// TIA Portal V20 export
DATA_BLOCK "IdentMvInterfaceHmi"   // DB219
// stored: InstanceOfName typeIdentMvHmi, InstanceOfType UDT
"typeIdentMvHmi"
   // VAR
   //    selectedUnit : USInt := 1;
   //    selectedEM : USInt;
   //    mvReaderId : USInt;
   //    numberOfMv : USInt;
   //    mvReader : Array[0.."NO_OF_MV_IDENT_DEVICES"] of "LSicar_typeIdentInterfaceHmi";
   // END_VAR
BEGIN
END_DATA_BLOCK
